Fanuc KAREL source: ko00033.KL

-- PROVISIONAL review KL for V1013-1; original PC SHA256 ee0791afb15266e702233c98287888f0fa36ba7b19c9d8a4b9900a08788f9df3
-- Incomplete behavior may be omitted. Consult companion uncertainty JSON. Do not deploy.
PROGRAM KO00033
%NOLOCKGROUP
BEGIN
  -- UNRESOLVED_PC offsets 5-12; opcodes 9D,23
  -- UNRESOLVED_PC offsets 17-66; opcodes 27,27,49,7E,AD,22,1C,22,31,7E,4A
  -- UNRESOLVED_PC offsets 71-75; opcodes 7F
END KO00033
